// TIA Portal project "Bibite" (V16)

(* hardware
DEVICE "S7-1200 station_1"  S7-1200 Station
   slot 0: "Telaio di montaggio_0"  S7-1200 Rack  Rack  V1.0
   slot 1: "PLC_1"  CPU 1214C DC/DC/DC  6ES7 214-1AG40-0XB0  V4.1
*)

// ===== PLC "PLC_1"  CPU 1214C DC/DC/DC =====

VAR_GLOBAL   // PLC tag table "Tabella delle variabili standard"
   "Moneta" AT %I0.0 : Bool;
   "FineCorsaA" AT %I0.1 : Bool;
   "FineCorsaB" AT %I0.2 : Bool;
   "BibitaPresente" AT %I0.3 : Bool;
   "Prelievo" AT %M0.0 : Bool;
   "SA" AT %Q0.0 : Bool;
   "SB" AT %Q0.1 : Bool;
   "BLOCCA" AT %Q0.2 : Bool;
END_VAR

VAR_GLOBAL CONSTANT   // PLC tag table "Tabella delle variabili standard"
   "Delay" : Time := T#5s;
END_VAR

DATA_BLOCK "VariabiliDiStato"   // DB1
{ S7_Optimized_Access := 'TRUE' }
VERSION : 0.1
   VAR RETAIN
      HOME : Bool := true;
      ConsegnaBibita : Bool;
      RientroSB : Bool;
      NuovaBibita : Bool;
      RientroSA : Bool;
      Attesa : Bool;
   END_VAR
BEGIN
END_DATA_BLOCK

// folder: System blocks/Program resources

DATA_BLOCK "IEC_Timer_0_DB"   // DB2
{ S7_Optimized_Access := 'TRUE' }
AUTHOR : Simatic
FAMILY : IEC
NAME : IEC_TMR
VERSION : 1.0
// stored: InstanceOfName IEC_TIMER
"IEC_TIMER"
BEGIN
END_DATA_BLOCK

DATA_BLOCK "IEC_Timer_0_DB_1"   // DB3
{ S7_Optimized_Access := 'TRUE' }
AUTHOR : Simatic
FAMILY : IEC
NAME : IEC_TMR
VERSION : 1.0
// stored: InstanceOfName IEC_TIMER
"IEC_TIMER"
BEGIN
END_DATA_BLOCK

// folder: (top level)

ORGANIZATION_BLOCK "Main"   // OB1, LAD, ProgramCycle
TITLE = "Main Program Sweep (Cycle)"
{ S7_Optimized_Access := 'TRUE' }
VERSION : 0.1
   VAR_INPUT
      Initial_Call : Bool;   // Initial call of this OB
      Remanence : Bool;   // =True, if remanent data are available
   END_VAR
BEGIN

REGION Network 1
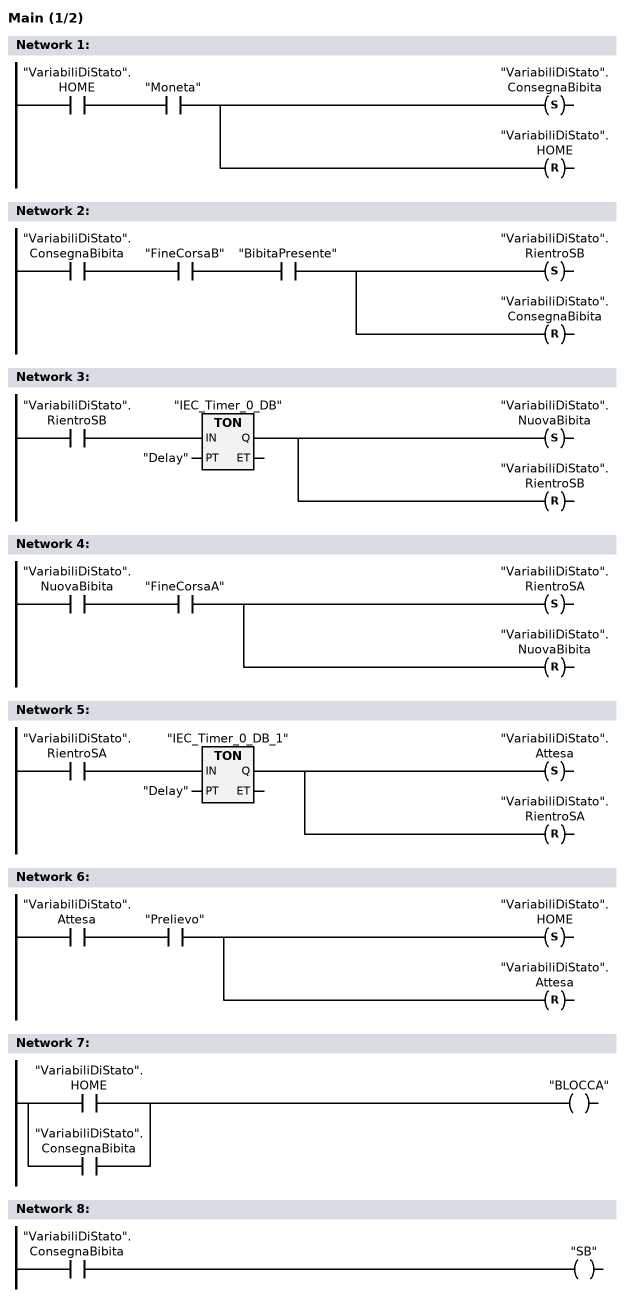
   RUNG wire#powerrail
      Contact( "VariabiliDiStato".HOME )
      Contact( "Moneta" )
      wire#w1
      S_Coil( "VariabiliDiStato".ConsegnaBibita )
   END_RUNG
   RUNG wire#w1
      R_Coil( "VariabiliDiStato".HOME )
   END_RUNG
   // the same network as SCL:
   IF "VariabiliDiStato".HOME AND "Moneta" THEN
       "VariabiliDiStato".ConsegnaBibita := TRUE;
       "VariabiliDiStato".HOME := FALSE;
   END_IF;
END_REGION

REGION Network 2
   RUNG wire#powerrail
      Contact( "VariabiliDiStato".ConsegnaBibita )
      Contact( "FineCorsaB" )
      Contact( "BibitaPresente" )
      wire#w1
      S_Coil( "VariabiliDiStato".RientroSB )
   END_RUNG
   RUNG wire#w1
      R_Coil( "VariabiliDiStato".ConsegnaBibita )
   END_RUNG
   // the same network as SCL:
   IF "VariabiliDiStato".ConsegnaBibita AND "FineCorsaB" AND "BibitaPresente" THEN
       "VariabiliDiStato".RientroSB := TRUE;
       "VariabiliDiStato".ConsegnaBibita := FALSE;
   END_IF;
END_REGION

REGION Network 3
   "IEC_Timer_0_DB".TON(IN := "VariabiliDiStato".RientroSB, PT := "Delay");
   IF "IEC_Timer_0_DB".Q THEN
       "VariabiliDiStato".NuovaBibita := TRUE;
       "VariabiliDiStato".RientroSB := FALSE;
   END_IF;
END_REGION

REGION Network 4
   RUNG wire#powerrail
      Contact( "VariabiliDiStato".NuovaBibita )
      Contact( "FineCorsaA" )
      wire#w1
      S_Coil( "VariabiliDiStato".RientroSA )
   END_RUNG
   RUNG wire#w1
      R_Coil( "VariabiliDiStato".NuovaBibita )
   END_RUNG
   // the same network as SCL:
   IF "VariabiliDiStato".NuovaBibita AND "FineCorsaA" THEN
       "VariabiliDiStato".RientroSA := TRUE;
       "VariabiliDiStato".NuovaBibita := FALSE;
   END_IF;
END_REGION

REGION Network 5
   "IEC_Timer_0_DB_1".TON(IN := "VariabiliDiStato".RientroSA, PT := "Delay");
   IF "IEC_Timer_0_DB_1".Q THEN
       "VariabiliDiStato".Attesa := TRUE;
       "VariabiliDiStato".RientroSA := FALSE;
   END_IF;
END_REGION

REGION Network 6
   RUNG wire#powerrail
      Contact( "VariabiliDiStato".Attesa )
      Contact( "Prelievo" )
      wire#w1
      S_Coil( "VariabiliDiStato".HOME )
   END_RUNG
   RUNG wire#w1
      R_Coil( "VariabiliDiStato".Attesa )
   END_RUNG
   // the same network as SCL:
   IF "VariabiliDiStato".Attesa AND "Prelievo" THEN
       "VariabiliDiStato".HOME := TRUE;
       "VariabiliDiStato".Attesa := FALSE;
   END_IF;
END_REGION

REGION Network 7
   RUNG wire#powerrail
      Contact( "VariabiliDiStato".HOME )
      wire#w1
      Coil( "BLOCCA" )
   END_RUNG
   RUNG wire#powerrail
      Contact( "VariabiliDiStato".ConsegnaBibita )
   END_RUNG wire#w1
   // the same network as SCL:
   "BLOCCA" := "VariabiliDiStato".HOME OR "VariabiliDiStato".ConsegnaBibita;
END_REGION

REGION Network 8
   RUNG wire#powerrail
      Contact( "VariabiliDiStato".ConsegnaBibita )
      Coil( "SB" )
   END_RUNG
   // the same network as SCL:
   "SB" := "VariabiliDiStato".ConsegnaBibita;
END_REGION

REGION Network 9
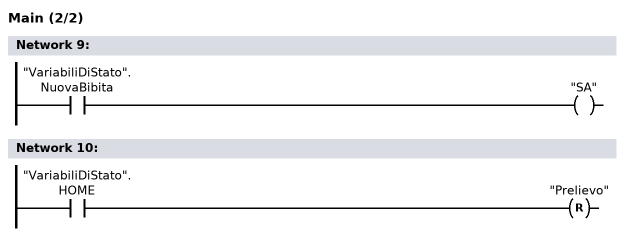
   RUNG wire#powerrail
      Contact( "VariabiliDiStato".NuovaBibita )
      Coil( "SA" )
   END_RUNG
   // the same network as SCL:
   "SA" := "VariabiliDiStato".NuovaBibita;
END_REGION

REGION Network 10
   RUNG wire#powerrail
      Contact( "VariabiliDiStato".HOME )
      R_Coil( "Prelievo" )
   END_RUNG
   // the same network as SCL:
   IF "VariabiliDiStato".HOME THEN "Prelievo" := FALSE; END_IF;
END_REGION
END_ORGANIZATION_BLOCK

ORGANIZATION_BLOCK "Hardware interrupt"   // OB40, LAD, HWProcessInterrupt
{ S7_Optimized_Access := 'TRUE' }
VERSION : 0.1
   VAR_INPUT
      LADDR : Hw_Io;   // Hardware identifier
      USI : Word;   // User structure identifier
      IChannel : USInt;   // Interrupt channel number
      EventType : Byte;   // EventType
   END_VAR
BEGIN

REGION Network 1
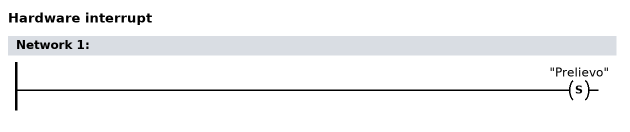
   RUNG wire#powerrail
      S_Coil( "Prelievo" )
   END_RUNG
   // the same network as SCL:
   "Prelievo" := TRUE;
END_REGION
END_ORGANIZATION_BLOCK